{attribute 'GeneratedUsingTerminal: EL6224-0000-0021'}
{attribute addProperty BoxType "EL6224-0000-0021"}
{attribute addProperty Id "DeviceState_Inputs_DeviceAT %I*DeviceState_Inputs_Device_A12105982DeviceState_InputsAT %I*DeviceState_Inputs_4751FF764IO_Link_Port1_inAT %I*IO_Link_Port1_in_4EEDF10D10IO_Link_Port2_inAT %I*IO_Link_Port2_in_4EEDF10D10IO_Link_Port3_inAT %I*IO_Link_Port3_in_4EEDF10D10IO_Link_Port4_inAT %I*IO_Link_Port4_in_4EEDF10D10IO_Link_Port1_outAT %Q*IO_Link_Port1_out_F2E0F4CF10IO_Link_Port2_outAT %Q*IO_Link_Port2_out_F2E0F4CF10IO_Link_Port3_outAT %Q*IO_Link_Port3_out_F2E0F4CF10IO_Link_Port4_outAT %Q*IO_Link_Port4_out_F2E0F4CF10WcStateAT %I*WcState_9091E0EB2InfoDataAT %I*InfoData_41C547A32"}
{attribute addProperty CRC "1128901421"}
{attribute addProperty Size "90"}
TYPE EL6224_4349AB2D EXTENDS EtcSlaveTerminalBase_947E5A46 :
STRUCT
	{attribute addProperty Name "DeviceState_Inputs_Device"}
	DeviceState_Inputs_Device : DeviceState_Inputs_Device_A1210598;
	{attribute addProperty Name "DeviceState_Inputs"}
	DeviceState_Inputs : DeviceState_Inputs_4751FF76;
	{attribute addProperty Name "IO_Link_Port1_in"}
	IO_Link_Port1_in : IO_Link_Port1_in_4EEDF10D;
	{attribute addProperty Name "IO_Link_Port2_in"}
	IO_Link_Port2_in : IO_Link_Port2_in_4EEDF10D;
	{attribute addProperty Name "IO_Link_Port3_in"}
	IO_Link_Port3_in : IO_Link_Port3_in_4EEDF10D;
	{attribute addProperty Name "IO_Link_Port4_in"}
	IO_Link_Port4_in : IO_Link_Port4_in_4EEDF10D;
	{attribute addProperty Name "IO_Link_Port1_out"}
	IO_Link_Port1_out : IO_Link_Port1_out_F2E0F4CF;
	{attribute addProperty Name "IO_Link_Port2_out"}
	IO_Link_Port2_out : IO_Link_Port2_out_F2E0F4CF;
	{attribute addProperty Name "IO_Link_Port3_out"}
	IO_Link_Port3_out : IO_Link_Port3_out_F2E0F4CF;
	{attribute addProperty Name "IO_Link_Port4_out"}
	IO_Link_Port4_out : IO_Link_Port4_out_F2E0F4CF;
	{attribute addProperty Name "WcState"}
	WcState : WcState_9091E0EB;
	{attribute addProperty Name "InfoData"}
	InfoData : InfoData_41C547A3;
END_STRUCT
END_TYPE

(* stored: Version 1.2.0.0, ProductVersion 3.1.4024.9
   DUT EL6224_4349AB2D: Id {cc22323e-72cd-40b3-bd38-a0bade2adf4d} *)
